// TIA Portal V18 export
FUNCTION_BLOCK "Alarms"   // FB18, LAD
{ S7_Optimized_Access := 'TRUE' }
// stored: AutoNumber false, MemoryReserve 100, SetENOAutomatically false
   VAR
      BypassTempAlarm_TON { S7_SetPoint := 'True'} : TON_TIME;
      TDPressTxFaul_TON { S7_SetPoint := 'True'} : TON_TIME;
      HiTemp_TON { S7_SetPoint := 'True'} : TON_TIME;
      NoFlushFlow_TON { S7_SetPoint := 'True'} : TON_TIME;
      ChargeFault_TON { S7_SetPoint := 'True'} : TON_TIME;
      HiTempRPM_TON { S7_SetPoint := 'True'} : TON_TIME;
      HornOn_TP { S7_SetPoint := 'True'} : TP_TIME;   // Time horn is on for when request come through
      HiTempAlarm_TON { S7_SetPoint := 'True'} : TON_TIME;
      FlushFault_TP { S7_SetPoint := 'True'} : TP_TIME;
      LubeFlowFault_TON { S7_SetPoint := 'True'} : TON_TIME;
      LubeFault_TP { S7_SetPoint := 'True'} : TP_TIME;
      Charge2Fault_TON { S7_SetPoint := 'True'} : TON_TIME;
      Charge1Fault_TP { S7_SetPoint := 'True'} : TP_TIME;
      Charge2Fault_TP { S7_SetPoint := 'True'} : TP_TIME;
      FilterFault_TP { S7_SetPoint := 'True'} : TP_TIME;
      AuxPumpFault_TP { S7_SetPoint := 'True'} : TP_TIME;
      FanFault_TP { S7_SetPoint := 'True'} : TP_TIME;
      M1Fault_TP { S7_SetPoint := 'True'} : TP_TIME;
      M2Fault_TP { S7_SetPoint := 'True'} : TP_TIME;
      HiTempFault_TP { S7_SetPoint := 'True'} : TP_TIME;
      TankLevelFault_TP { S7_SetPoint := 'True'} : TP_TIME;
      TankTempFault_TP { S7_SetPoint := 'True'} : TP_TIME;
      HiTempShtdwn_TP { S7_SetPoint := 'True'} : TP_TIME;
      TDPressTXFault_TP { S7_SetPoint := 'True'} : TP_TIME;
      EngineFault_TP { S7_SetPoint := 'True'} : TP_TIME;
      BypassHiTemp_Tp { S7_SetPoint := 'True'} : TP_TIME;
      ComFault_Tp { S7_SetPoint := 'True'} : TP_TIME;
      SystemFault_Tp { S7_SetPoint := 'True'} : TP_TIME;
   END_VAR
   VAR_TEMP
      tempReal : Real;
      tempBool : Bool;
      tempTime : Time;
   END_VAR
   VAR_TEMP   // added for the SCL form of the ladder/FBD networks
      _w1 : Bool;
      _w2 : Bool;
   END_VAR
BEGIN

REGION Network 1: TD Flush Fault
   // If Aux Pump running and not in Hand and no flush within in set time disable spin
   // Aux Pump in Hand is Bypass for no flush interlock
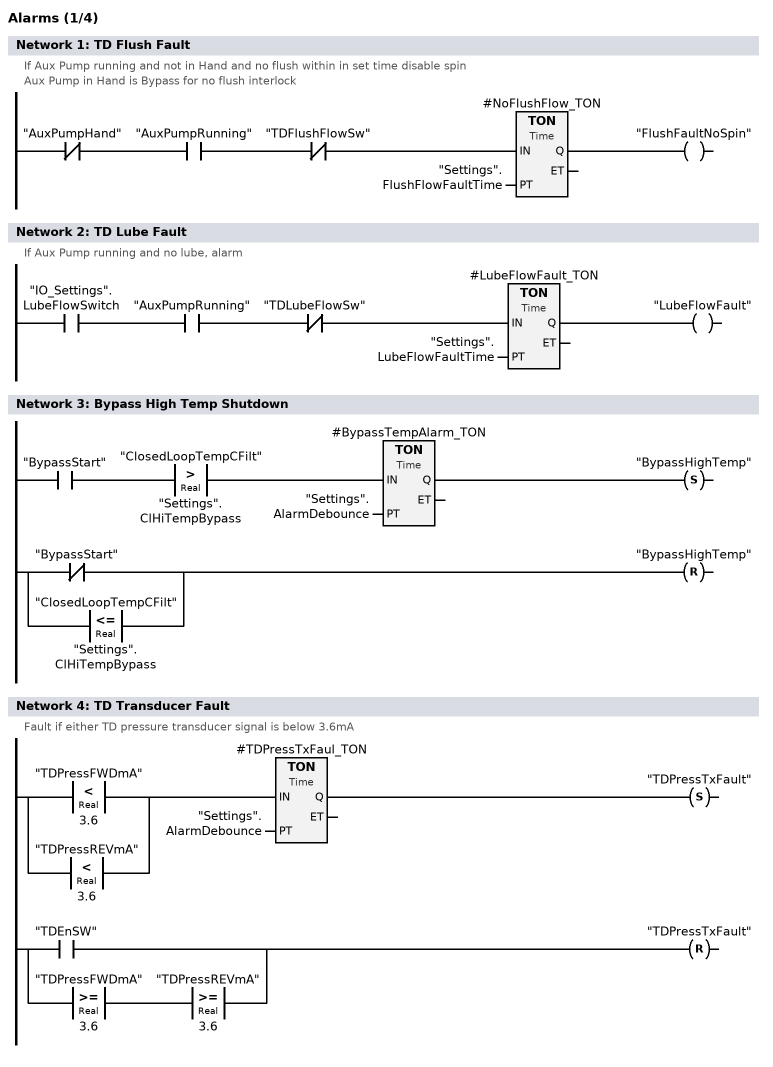
   RUNG wire#powerrail
      I_Contact( "AuxPumpHand" )
      Contact( "AuxPumpRunning" )
      I_Contact( "TDFlushFlowSw" )
      { S7_Templates := "time_type := Time" } #NoFlushFlow_TON.TON(pt := "Settings".FlushFlowFaultTime, et =>)
      Coil( "FlushFaultNoSpin" )
   END_RUNG
   // the same network as SCL:
   #NoFlushFlow_TON(IN := NOT "AuxPumpHand" AND "AuxPumpRunning" AND NOT "TDFlushFlowSw",   // TON
                    PT := "Settings".FlushFlowFaultTime);
   "FlushFaultNoSpin" := #NoFlushFlow_TON.Q;
END_REGION

REGION Network 2: TD Lube Fault
   // If Aux Pump running and no lube, alarm
   RUNG wire#powerrail
      Contact( "IO_Settings".LubeFlowSwitch )
      Contact( "AuxPumpRunning" )
      I_Contact( "TDLubeFlowSw" )
      { S7_Templates := "time_type := Time" } #LubeFlowFault_TON.TON(pt := "Settings".LubeFlowFaultTime, et =>)
      Coil( "LubeFlowFault" )
   END_RUNG
   // the same network as SCL:
   #LubeFlowFault_TON(IN := "IO_Settings".LubeFlowSwitch AND "AuxPumpRunning" AND NOT "TDLubeFlowSw",   // TON
                      PT := "Settings".LubeFlowFaultTime);
   "LubeFlowFault" := #LubeFlowFault_TON.Q;
END_REGION

REGION Network 3: Bypass High Temp Shutdown
   RUNG wire#powerrail
      Contact( "BypassStart" )
      { S7_Templates := "SrcType := Real" } GT_Contact(in1 := "ClosedLoopTempCFilt", in2 := "Settings".ClHiTempBypass)
      { S7_Templates := "time_type := Time" } #BypassTempAlarm_TON.TON(pt := "Settings".AlarmDebounce, et =>)
      S_Coil( "BypassHighTemp" )
   END_RUNG
   RUNG wire#powerrail
      I_Contact( "BypassStart" )
      wire#w1
      R_Coil( "BypassHighTemp" )
   END_RUNG
   RUNG wire#powerrail
      { S7_Templates := "SrcType := Real" } LE_Contact(in1 := "ClosedLoopTempCFilt", in2 := "Settings".ClHiTempBypass)
   END_RUNG wire#w1
   // the same network as SCL:
   #BypassTempAlarm_TON(IN := "BypassStart" AND ("ClosedLoopTempCFilt" > "Settings".ClHiTempBypass),   // TON
                        PT := "Settings".AlarmDebounce);
   IF #BypassTempAlarm_TON.Q THEN "BypassHighTemp" := TRUE; END_IF;
   IF NOT "BypassStart" OR ("ClosedLoopTempCFilt" <= "Settings".ClHiTempBypass) THEN
       "BypassHighTemp" := FALSE;
   END_IF;
END_REGION

REGION Network 4: TD Transducer Fault
   // Fault if either TD pressure transducer signal is below 3.6mA
   RUNG wire#powerrail
      { S7_Templates := "SrcType := Real" } LT_Contact(in1 := "TDPressFWDmA", in2 := 3.6)
      wire#w1
      { S7_Templates := "time_type := Time" } #TDPressTxFaul_TON.TON(pt := "Settings".AlarmDebounce, et =>)
      S_Coil( "TDPressTxFault" )
   END_RUNG
   RUNG wire#powerrail
      { S7_Templates := "SrcType := Real" } LT_Contact(in1 := "TDPressREVmA", in2 := 3.6)
   END_RUNG wire#w1
   RUNG wire#powerrail
      Contact( "TDEnSW" )
      wire#w2
      R_Coil( "TDPressTxFault" )
   END_RUNG
   RUNG wire#powerrail
      { S7_Templates := "SrcType := Real" } GE_Contact(in1 := "TDPressFWDmA", in2 := 3.6)
      { S7_Templates := "SrcType := Real" } GE_Contact(in1 := "TDPressREVmA", in2 := 3.6)
   END_RUNG wire#w2
   // the same network as SCL:
   #TDPressTxFaul_TON(IN := ("TDPressFWDmA" < 3.6) OR ("TDPressREVmA" < 3.6), PT := "Settings".AlarmDebounce);   // TON
   IF #TDPressTxFaul_TON.Q THEN "TDPressTxFault" := TRUE; END_IF;
   IF "TDEnSW" OR (("TDPressFWDmA" >= 3.6) AND ("TDPressREVmA" >= 3.6)) THEN
       "TDPressTxFault" := FALSE;
   END_IF;
END_REGION

REGION Network 5: Closed Loop High Temp Shutdown
   // Reduce RPM if temp above RPM reduction temp
   // Shudown if temp above shutdown.
   // Reset either when 3 C below trigger point
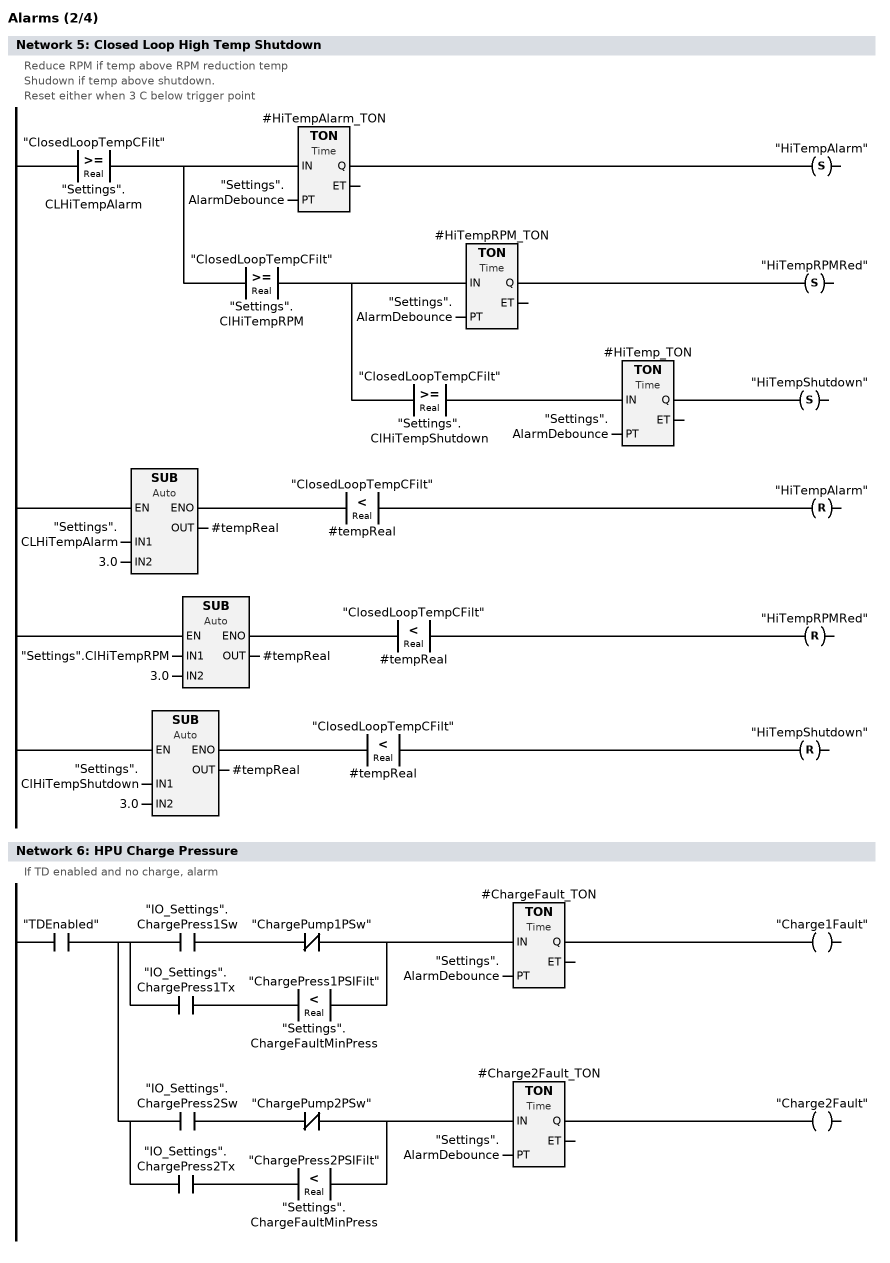
   RUNG wire#powerrail
      { S7_Templates := "SrcType := Real" } GE_Contact(in1 := "ClosedLoopTempCFilt", in2 := "Settings".CLHiTempAlarm)
      wire#w1
      { S7_Templates := "time_type := Time" } #HiTempAlarm_TON.TON(pt := "Settings".AlarmDebounce, et =>)
      S_Coil( "HiTempAlarm" )
   END_RUNG
   RUNG wire#w1
      { S7_Templates := "SrcType := Real" } GE_Contact(in1 := "ClosedLoopTempCFilt", in2 := "Settings".ClHiTempRPM)
      wire#w2
      { S7_Templates := "time_type := Time" } #HiTempRPM_TON.TON(pt := "Settings".AlarmDebounce, et =>)
      S_Coil( "HiTempRPMRed" )
   END_RUNG
   RUNG wire#w2
      { S7_Templates := "SrcType := Real" } GE_Contact(in1 := "ClosedLoopTempCFilt", in2 := "Settings".ClHiTempShutdown)
      { S7_Templates := "time_type := Time" } #HiTemp_TON.TON(pt := "Settings".AlarmDebounce, et =>)
      S_Coil( "HiTempShutdown" )
   END_RUNG
   RUNG wire#powerrail
      Sub(in1 := "Settings".CLHiTempAlarm, in2 := 3.0, out => #tempReal)
      { S7_Templates := "SrcType := Real" } LT_Contact(in1 := "ClosedLoopTempCFilt", in2 := #tempReal)
      R_Coil( "HiTempAlarm" )
   END_RUNG
   RUNG wire#powerrail
      Sub(in1 := "Settings".ClHiTempRPM, in2 := 3.0, out => #tempReal)
      { S7_Templates := "SrcType := Real" } LT_Contact(in1 := "ClosedLoopTempCFilt", in2 := #tempReal)
      R_Coil( "HiTempRPMRed" )
   END_RUNG
   RUNG wire#powerrail
      Sub(in1 := "Settings".ClHiTempShutdown, in2 := 3.0, out => #tempReal)
      { S7_Templates := "SrcType := Real" } LT_Contact(in1 := "ClosedLoopTempCFilt", in2 := #tempReal)
      R_Coil( "HiTempShutdown" )
   END_RUNG
   // the same network as SCL:
   #_w1 := "ClosedLoopTempCFilt" >= "Settings".CLHiTempAlarm;
   #HiTempAlarm_TON(IN := #_w1, PT := "Settings".AlarmDebounce);   // TON
   IF #HiTempAlarm_TON.Q THEN "HiTempAlarm" := TRUE; END_IF;
   #_w2 := #_w1 AND ("ClosedLoopTempCFilt" >= "Settings".ClHiTempRPM);
   #HiTempRPM_TON(IN := #_w2, PT := "Settings".AlarmDebounce);   // TON
   IF #HiTempRPM_TON.Q THEN "HiTempRPMRed" := TRUE; END_IF;
   #HiTemp_TON(IN := #_w2 AND ("ClosedLoopTempCFilt" >= "Settings".ClHiTempShutdown),   // TON
               PT := "Settings".AlarmDebounce);
   IF #HiTemp_TON.Q THEN "HiTempShutdown" := TRUE; END_IF;
   #tempReal := "Settings".CLHiTempAlarm - 3.0;
   IF "ClosedLoopTempCFilt" < #tempReal THEN "HiTempAlarm" := FALSE; END_IF;
   #tempReal := "Settings".ClHiTempRPM - 3.0;
   IF "ClosedLoopTempCFilt" < #tempReal THEN "HiTempRPMRed" := FALSE; END_IF;
   #tempReal := "Settings".ClHiTempShutdown - 3.0;
   IF "ClosedLoopTempCFilt" < #tempReal THEN "HiTempShutdown" := FALSE; END_IF;
END_REGION

REGION Network 6: HPU Charge Pressure
   // If TD enabled and no charge, alarm
   RUNG wire#powerrail
      Contact( "TDEnabled" )
      wire#w1
      Contact( "IO_Settings".ChargePress1Sw )
      I_Contact( "ChargePump1PSw" )
      wire#w2
      { S7_Templates := "time_type := Time" } #ChargeFault_TON.TON(pt := "Settings".AlarmDebounce, et =>)
      Coil( "Charge1Fault" )
   END_RUNG
   RUNG wire#w1
      Contact( "IO_Settings".ChargePress1Tx )
      { S7_Templates := "SrcType := Real" } LT_Contact(in1 := "ChargePress1PSIFilt", in2 := "Settings".ChargeFaultMinPress)
   END_RUNG wire#w2
   RUNG wire#w1
      Contact( "IO_Settings".ChargePress2Sw )
      I_Contact( "ChargePump2PSw" )
      wire#w3
      { S7_Templates := "time_type := Time" } #Charge2Fault_TON.TON(pt := "Settings".AlarmDebounce, et =>)
      Coil( "Charge2Fault" )
   END_RUNG
   RUNG wire#w1
      Contact( "IO_Settings".ChargePress2Tx )
      { S7_Templates := "SrcType := Real" } LT_Contact(in1 := "ChargePress2PSIFilt", in2 := "Settings".ChargeFaultMinPress)
   END_RUNG wire#w3
   // the same network as SCL:
   #ChargeFault_TON(IN := "TDEnabled" AND (("IO_Settings".ChargePress1Sw AND NOT "ChargePump1PSw") OR ("IO_Settings".ChargePress1Tx AND ("ChargePress1PSIFilt" < "Settings".ChargeFaultMinPress))),   // TON
                    PT := "Settings".AlarmDebounce);
   "Charge1Fault" := #ChargeFault_TON.Q;
   #Charge2Fault_TON(IN := "TDEnabled" AND (("IO_Settings".ChargePress2Sw AND NOT "ChargePump2PSw") OR ("IO_Settings".ChargePress2Tx AND ("ChargePress2PSIFilt" < "Settings".ChargeFaultMinPress))),   // TON
                     PT := "Settings".AlarmDebounce);
   "Charge2Fault" := #Charge2Fault_TON.Q;
END_REGION

REGION Network 7: Plug Filter
   // Set if any filter is plugged or charge above 1000
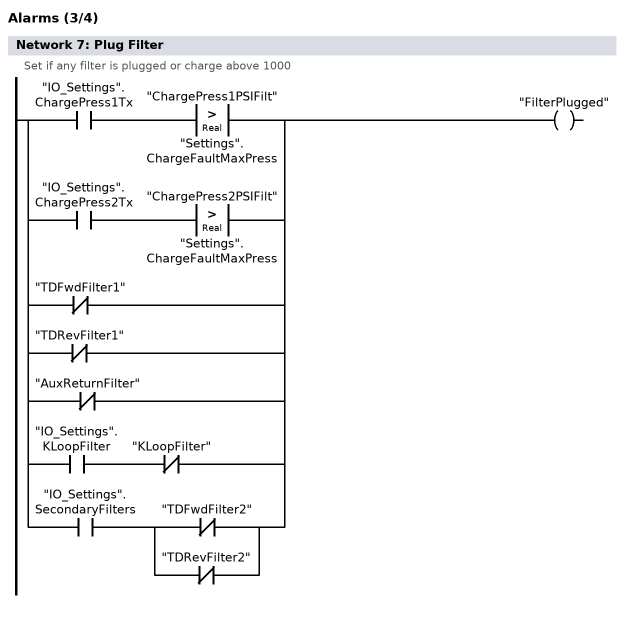
   RUNG wire#powerrail
      Contact( "IO_Settings".ChargePress1Tx )
      { S7_Templates := "SrcType := Real" } GT_Contact(in1 := "ChargePress1PSIFilt", in2 := "Settings".ChargeFaultMaxPress)
      wire#w1
      Coil( "FilterPlugged" )
   END_RUNG
   RUNG wire#powerrail
      Contact( "IO_Settings".ChargePress2Tx )
      { S7_Templates := "SrcType := Real" } GT_Contact(in1 := "ChargePress2PSIFilt", in2 := "Settings".ChargeFaultMaxPress)
   END_RUNG wire#w1
   RUNG wire#powerrail
      I_Contact( "TDFwdFilter1" )
   END_RUNG wire#w1
   RUNG wire#powerrail
      I_Contact( "TDRevFilter1" )
   END_RUNG wire#w1
   RUNG wire#powerrail
      I_Contact( "AuxReturnFilter" )
   END_RUNG wire#w1
   RUNG wire#powerrail
      Contact( "IO_Settings".KLoopFilter )
      I_Contact( "KLoopFilter" )
   END_RUNG wire#w1
   RUNG wire#powerrail
      Contact( "IO_Settings".SecondaryFilters )
      wire#w2
      I_Contact( "TDFwdFilter2" )
   END_RUNG wire#w1
   RUNG wire#w2
      I_Contact( "TDRevFilter2" )
   END_RUNG wire#w1
   // the same network as SCL:
   "FilterPlugged" := ("IO_Settings".ChargePress1Tx AND ("ChargePress1PSIFilt" > "Settings".ChargeFaultMaxPress)) OR ("IO_Settings".ChargePress2Tx AND ("ChargePress2PSIFilt" > "Settings".ChargeFaultMaxPress)) OR NOT "TDFwdFilter1" OR NOT "TDRevFilter1" OR NOT "AuxReturnFilter" OR ("IO_Settings".KLoopFilter AND NOT "KLoopFilter") OR ("IO_Settings".SecondaryFilters AND (NOT "TDFwdFilter2" OR NOT "TDRevFilter2"));
END_REGION

REGION Network 8: Horn
   // Turn on Horn if test or
   // Sequence Pulse for horn time if any of following faults have a pulsed:
   // FlushFault/Low Level/Tank Temp/LubeFault/FilterPlugged/Any Motor Start Fault/Charge Pressure fault, engine fault.
   // Clock Horn for High Temp unless silenced
   // Trigger horn 1 a minute if reduced RPM.
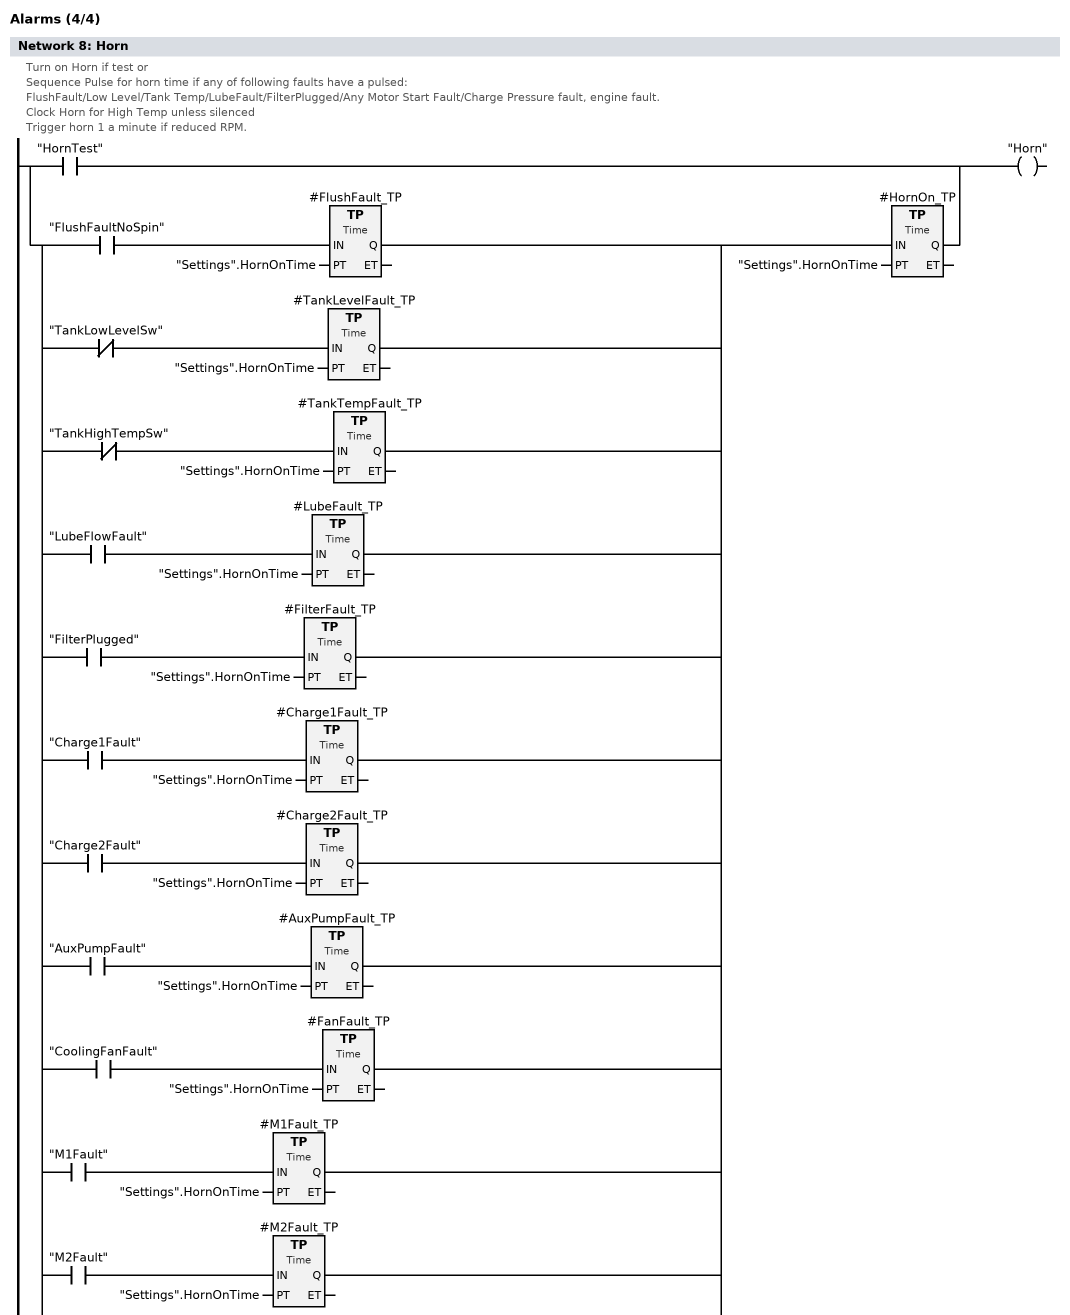
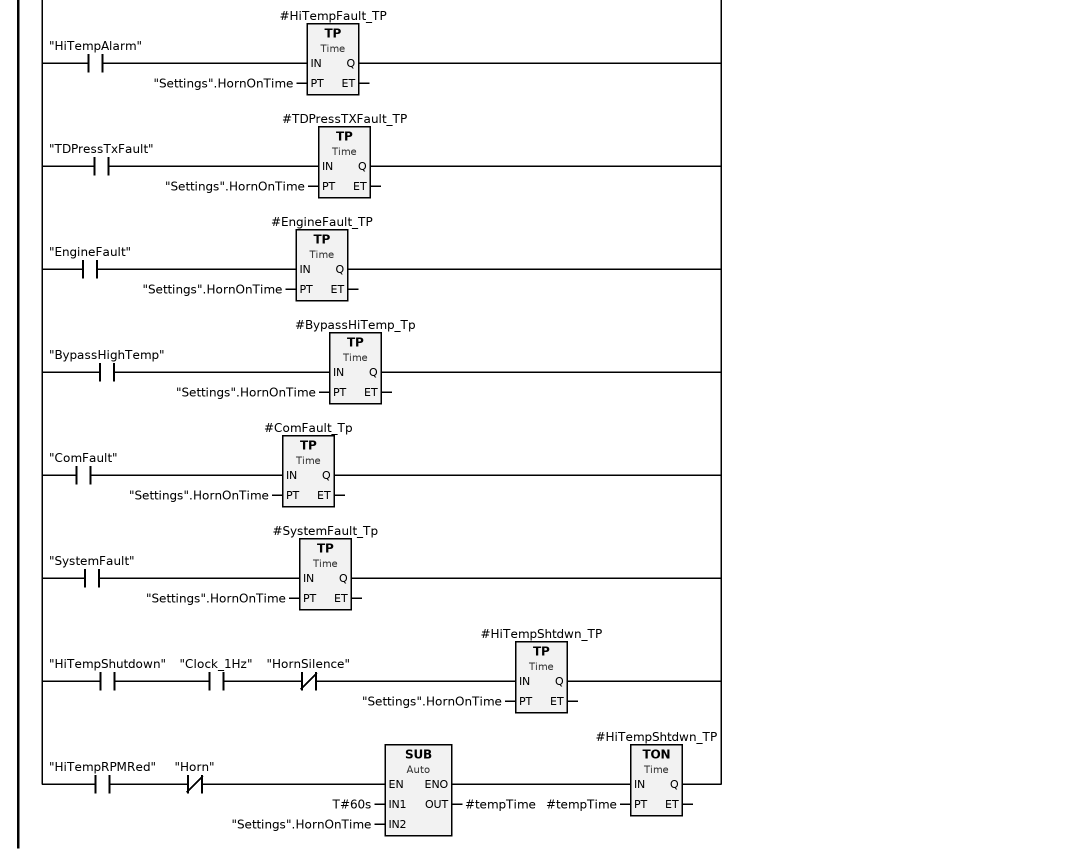
   RUNG wire#powerrail
      Contact( "HornTest" )
      wire#w1
      Coil( "Horn" )
   END_RUNG
   RUNG wire#powerrail
      Contact( "FlushFaultNoSpin" )
      { S7_Templates := "time_type := Time" } #FlushFault_TP.TP(pt := "Settings".HornOnTime, et =>)
      wire#w2
      { S7_Templates := "time_type := Time" } #HornOn_TP.TP(pt := "Settings".HornOnTime, et =>)
   END_RUNG wire#w1
   RUNG wire#powerrail
      I_Contact( "TankLowLevelSw" )
      { S7_Templates := "time_type := Time" } #TankLevelFault_TP.TP(pt := "Settings".HornOnTime, et =>)
   END_RUNG wire#w2
   RUNG wire#powerrail
      I_Contact( "TankHighTempSw" )
      { S7_Templates := "time_type := Time" } #TankTempFault_TP.TP(pt := "Settings".HornOnTime, et =>)
   END_RUNG wire#w2
   RUNG wire#powerrail
      Contact( "LubeFlowFault" )
      { S7_Templates := "time_type := Time" } #LubeFault_TP.TP(pt := "Settings".HornOnTime, et =>)
   END_RUNG wire#w2
   RUNG wire#powerrail
      Contact( "FilterPlugged" )
      { S7_Templates := "time_type := Time" } #FilterFault_TP.TP(pt := "Settings".HornOnTime, et =>)
   END_RUNG wire#w2
   RUNG wire#powerrail
      Contact( "Charge1Fault" )
      { S7_Templates := "time_type := Time" } #Charge1Fault_TP.TP(pt := "Settings".HornOnTime, et =>)
   END_RUNG wire#w2
   RUNG wire#powerrail
      Contact( "Charge2Fault" )
      { S7_Templates := "time_type := Time" } #Charge2Fault_TP.TP(pt := "Settings".HornOnTime, et =>)
   END_RUNG wire#w2
   RUNG wire#powerrail
      Contact( "AuxPumpFault" )
      { S7_Templates := "time_type := Time" } #AuxPumpFault_TP.TP(pt := "Settings".HornOnTime, et =>)
   END_RUNG wire#w2
   RUNG wire#powerrail
      Contact( "CoolingFanFault" )
      { S7_Templates := "time_type := Time" } #FanFault_TP.TP(pt := "Settings".HornOnTime, et =>)
   END_RUNG wire#w2
   RUNG wire#powerrail
      Contact( "M1Fault" )
      { S7_Templates := "time_type := Time" } #M1Fault_TP.TP(pt := "Settings".HornOnTime, et =>)
   END_RUNG wire#w2
   RUNG wire#powerrail
      Contact( "M2Fault" )
      { S7_Templates := "time_type := Time" } #M2Fault_TP.TP(pt := "Settings".HornOnTime, et =>)
   END_RUNG wire#w2
   RUNG wire#powerrail
      Contact( "HiTempAlarm" )
      { S7_Templates := "time_type := Time" } #HiTempFault_TP.TP(pt := "Settings".HornOnTime, et =>)
   END_RUNG wire#w2
   RUNG wire#powerrail
      Contact( "TDPressTxFault" )
      { S7_Templates := "time_type := Time" } #TDPressTXFault_TP.TP(pt := "Settings".HornOnTime, et =>)
   END_RUNG wire#w2
   RUNG wire#powerrail
      Contact( "EngineFault" )
      { S7_Templates := "time_type := Time" } #EngineFault_TP.TP(pt := "Settings".HornOnTime, et =>)
   END_RUNG wire#w2
   RUNG wire#powerrail
      Contact( "BypassHighTemp" )
      { S7_Templates := "time_type := Time" } #BypassHiTemp_Tp.TP(pt := "Settings".HornOnTime, et =>)
   END_RUNG wire#w2
   RUNG wire#powerrail
      Contact( "ComFault" )
      { S7_Templates := "time_type := Time" } #ComFault_Tp.TP(pt := "Settings".HornOnTime, et =>)
   END_RUNG wire#w2
   RUNG wire#powerrail
      Contact( "SystemFault" )
      { S7_Templates := "time_type := Time" } #SystemFault_Tp.TP(pt := "Settings".HornOnTime, et =>)
   END_RUNG wire#w2
   RUNG wire#powerrail
      Contact( "HiTempShutdown" )
      Contact( "Clock_1Hz" )
      I_Contact( "HornSilence" )
      { S7_Templates := "time_type := Time" } #HiTempShtdwn_TP.TP(pt := "Settings".HornOnTime, et =>)
   END_RUNG wire#w2
   RUNG wire#powerrail
      Contact( "HiTempRPMRed" )
      I_Contact( "Horn" )
      Sub(in1 := T#60s, in2 := "Settings".HornOnTime, out => #tempTime)
      { S7_Templates := "time_type := Time" } #HiTempShtdwn_TP.TON(pt := #tempTime, et =>)
   END_RUNG wire#w2
   // the same network as SCL:
   #FlushFault_TP(IN := "FlushFaultNoSpin", PT := "Settings".HornOnTime);   // TP
   #TankLevelFault_TP(IN := NOT "TankLowLevelSw", PT := "Settings".HornOnTime);   // TP
   #TankTempFault_TP(IN := NOT "TankHighTempSw", PT := "Settings".HornOnTime);   // TP
   #LubeFault_TP(IN := "LubeFlowFault", PT := "Settings".HornOnTime);   // TP
   #FilterFault_TP(IN := "FilterPlugged", PT := "Settings".HornOnTime);   // TP
   #Charge1Fault_TP(IN := "Charge1Fault", PT := "Settings".HornOnTime);   // TP
   #Charge2Fault_TP(IN := "Charge2Fault", PT := "Settings".HornOnTime);   // TP
   #AuxPumpFault_TP(IN := "AuxPumpFault", PT := "Settings".HornOnTime);   // TP
   #FanFault_TP(IN := "CoolingFanFault", PT := "Settings".HornOnTime);   // TP
   #M1Fault_TP(IN := "M1Fault", PT := "Settings".HornOnTime);   // TP
   #M2Fault_TP(IN := "M2Fault", PT := "Settings".HornOnTime);   // TP
   #HiTempFault_TP(IN := "HiTempAlarm", PT := "Settings".HornOnTime);   // TP
   #TDPressTXFault_TP(IN := "TDPressTxFault", PT := "Settings".HornOnTime);   // TP
   #EngineFault_TP(IN := "EngineFault", PT := "Settings".HornOnTime);   // TP
   #BypassHiTemp_Tp(IN := "BypassHighTemp", PT := "Settings".HornOnTime);   // TP
   #ComFault_Tp(IN := "ComFault", PT := "Settings".HornOnTime);   // TP
   #SystemFault_Tp(IN := "SystemFault", PT := "Settings".HornOnTime);   // TP
   #HiTempShtdwn_TP(IN := "HiTempShutdown" AND "Clock_1Hz" AND NOT "HornSilence", PT := "Settings".HornOnTime);   // TP
   #_w1 := "HiTempRPMRed" AND NOT "Horn";
   IF #_w1 THEN #tempTime := T#60s - "Settings".HornOnTime; END_IF;
   #_w2 := #HiTempShtdwn_TP.Q;
   #HiTempShtdwn_TP(IN := #_w1, PT := #tempTime);   // TON
   #HornOn_TP(IN := #FlushFault_TP.Q OR #TankLevelFault_TP.Q OR #TankTempFault_TP.Q OR #LubeFault_TP.Q OR #FilterFault_TP.Q OR #Charge1Fault_TP.Q OR #Charge2Fault_TP.Q OR #AuxPumpFault_TP.Q OR #FanFault_TP.Q OR #M1Fault_TP.Q OR #M2Fault_TP.Q OR #HiTempFault_TP.Q OR #TDPressTXFault_TP.Q OR #EngineFault_TP.Q OR #BypassHiTemp_Tp.Q OR #ComFault_Tp.Q OR #SystemFault_Tp.Q OR #_w2 OR #HiTempShtdwn_TP.Q,   // TP
              PT := "Settings".HornOnTime);
   "Horn" := "HornTest" OR #HornOn_TP.Q;
END_REGION
END_FUNCTION_BLOCK
